(* Logix 5000 project; controller Hose_HP_Test_Rig_V1 vendor 1 type 14 code 149 rev 32.11; software revision 32.00 *)
// Hose HP Test Rig - 4 Station

TASK MainTask (continuous, watchdog 500 ms) : MainProgram

MODULES
   Local : vendor 1 type 14 code 149 (Compact 0, rev 32.11)
       : 1769-IQ32 (Compact 2, rev 3.1, Input RPI 20 ms)
      Discrete_IO : Embedded (Compact 1, rev 3.1, Output RPI 20 ms)
       : vendor 1 type 7 code 73 (Compact 3, rev 3.1, Output RPI 20 ms)
       : 1769-IF8 (Compact 5, rev 1.1, Output RPI 80 ms)
       : 1769-IF8 (Compact 4, rev 1.1, Output RPI 80 ms)
      VERIFYPLC : vendor 1 type 14 code 196 (Ethernet 192.168.4.180, rev 32.1, $d488c7ae$ RPI 20 ms, $26341d39$ RPI 20 ms, $f5226f78$ RPI 20 ms, $c4b3cc1b$ RPI 20 ms, $dea25812$ RPI 20 ms, $98b97a8d$ RPI 20 ms, $11873bfc$ RPI 20 ms, $408f890f$ RPI 20 ms, $f2f849b6$ RPI 20 ms, $8edf7c21$ RPI 20 ms, $0545c3c0$ RPI 20 ms, $be141c43$ RPI 20 ms, $2e1c7de5$ RPI 20 ms, $86533d27$ RPI 20 ms, $ac6396f9$ RPI 20 ms, $0a9383db$ RPI 20 ms)
      REM : vendor 1534 type 12 code 8 (Ethernet 192.168.4.224, rev 1.1, StandardDataDriven RPI 5 ms)
END_MODULES

ADD_ON_INSTRUCTION BOTTOM_DECLAMP   (* revision 1.0 *)
VAR_INPUT
   SET_SEQ_NO : DINT; {required}
END_VAR
VAR_IN_OUT
   CUR_SEQ_NO : DINT; {required}
END_VAR
VAR_OUTPUT
   BOTTOM_DECLAMP_AUTO : BOOL; {required}
END_VAR
VAR_INPUT
   BOTTOM_CLAMP_PS : BOOL; {required}
END_VAR
VAR_OUTPUT
   BOTTOM_DECLAMP_OK : BOOL; {required}
END_VAR
VAR_INPUT
   BOTTOM_NOT_DECLAMPED : BOOL; {required}
   FAULTED : BOOL; {required}
   RST_SEQ_ON : BOOL; {required}
   NEXT_SEQ_NO : DINT; {required}
END_VAR
VAR
   BOTTOM_DECLAMP_SEQ_AUTO : BOOL; {access None}
   ONS1 : BOOL; {access None}
   BOTTOM_DECLAMP_CHK_DEL : TIMER := (PRE := 500); {access None}
END_VAR

ROUTINE Logic   (* ladder *)
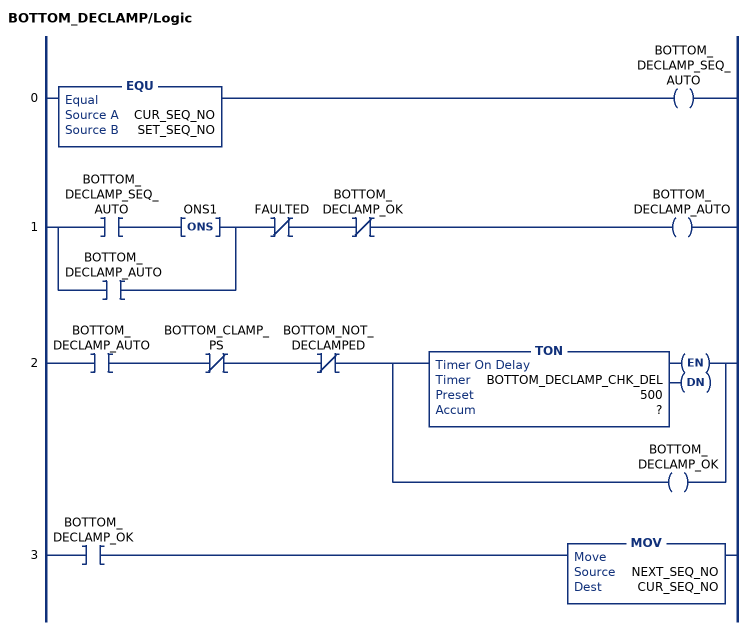
   0: EQU(CUR_SEQ_NO,SET_SEQ_NO)OTE(BOTTOM_DECLAMP_SEQ_AUTO);
   1: [XIC(BOTTOM_DECLAMP_SEQ_AUTO) ONS(ONS1) ,XIC(BOTTOM_DECLAMP_AUTO) ]XIO(FAULTED)XIO(BOTTOM_DECLAMP_OK)OTE(BOTTOM_DECLAMP_AUTO);
   2: XIC(BOTTOM_DECLAMP_AUTO)XIO(BOTTOM_CLAMP_PS)XIO(BOTTOM_NOT_DECLAMPED)[TON(BOTTOM_DECLAMP_CHK_DEL,?,?) ,OTE(BOTTOM_DECLAMP_OK) ];
   3: XIC(BOTTOM_DECLAMP_OK)MOV(NEXT_SEQ_NO,CUR_SEQ_NO);
END_ROUTINE
END_ADD_ON_INSTRUCTION

ADD_ON_INSTRUCTION CLAMP_FAULT   (* revision 1.0 *)
VAR_INPUT
   CLAMP_PR_SEL : BOOL; {required}
   CLAMP_PR_CHK : BOOL; {required}
   CLAMP_PR : DINT; {required}
   CLAMP_2BAR_LL : REAL; {required}
   CLAMP_2BAR_HL : REAL; {required}
   CLAMP_4BAR_LL : REAL; {required}
   CLAMP_4BAR_HL : REAL; {required}
   FLT_CLR_ONS : BOOL; {required}
END_VAR
VAR_OUTPUT
   CLAMP_2BPR_LOW : BOOL; {access Read Only, required}
   CLAMP_2BPR_HIGH : BOOL; {access Read Only, required}
   CLAMP_4BPR_LOW : BOOL; {access Read Only, required}
   CLAMP_4BPR_HIGH : BOOL; {access Read Only, required}
END_VAR
VAR_IN_OUT
   MSG : DINT; {required}
END_VAR

ROUTINE Logic   (* ladder *)
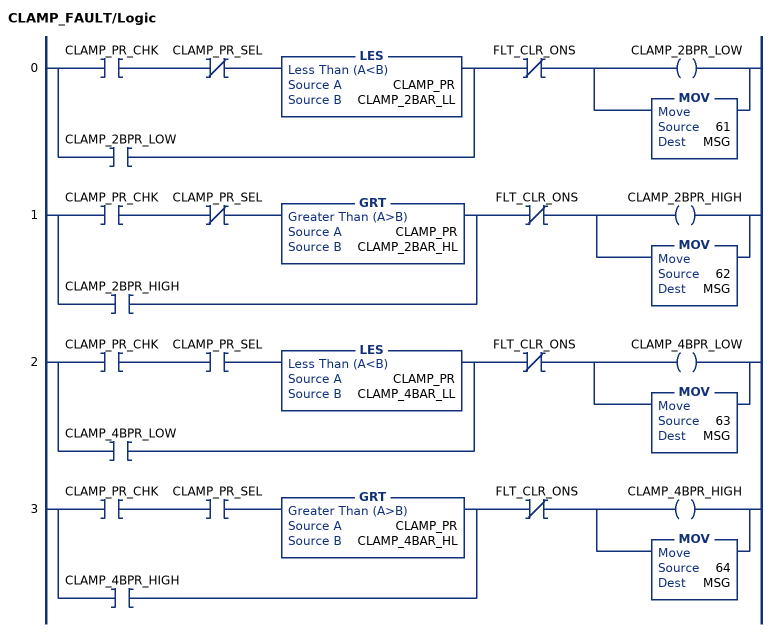
   0: [XIC(CLAMP_PR_CHK) XIO(CLAMP_PR_SEL) LES(CLAMP_PR,CLAMP_2BAR_LL) ,XIC(CLAMP_2BPR_LOW) ]XIO(FLT_CLR_ONS)[OTE(CLAMP_2BPR_LOW) ,MOV(61,MSG) ];
   1: [XIC(CLAMP_PR_CHK) XIO(CLAMP_PR_SEL) GRT(CLAMP_PR,CLAMP_2BAR_HL) ,XIC(CLAMP_2BPR_HIGH) ]XIO(FLT_CLR_ONS)[OTE(CLAMP_2BPR_HIGH) ,MOV(62,MSG) ];
   2: [XIC(CLAMP_PR_CHK) XIC(CLAMP_PR_SEL) LES(CLAMP_PR,CLAMP_4BAR_LL) ,XIC(CLAMP_4BPR_LOW) ]XIO(FLT_CLR_ONS)[OTE(CLAMP_4BPR_LOW) ,MOV(63,MSG) ];
   3: [XIC(CLAMP_PR_CHK) XIC(CLAMP_PR_SEL) GRT(CLAMP_PR,CLAMP_4BAR_HL) ,XIC(CLAMP_4BPR_HIGH) ]XIO(FLT_CLR_ONS)[OTE(CLAMP_4BPR_HIGH) ,MOV(64,MSG) ];
END_ROUTINE
END_ADD_ON_INSTRUCTION

ADD_ON_INSTRUCTION CONSTRICTION_FILL_OFF_SEQ   (* revision 1.0 *)
VAR_INPUT
   SET_SEQ_NO : DINT; {required}
END_VAR
VAR_IN_OUT
   CURR_SEQ_NO : DINT; {required}
END_VAR
VAR_INPUT
   TEST_ON : BOOL; {required}
END_VAR
VAR_OUTPUT
   CFILL_VAL_OFF : BOOL; {required}
   EXHS_VAL_OFF : BOOL; {required}
END_VAR
VAR_INPUT
   FAULTED : BOOL; {required}
   RST_SEQ_ON : BOOL; {required}
   NEXT_SEQ_NO : DINT; {required}
END_VAR
VAR
   SEQ_START : BOOL; {access None}
   ONS1 : BOOL; {access None}
   CFILL_VAL_OFF_DEL : TIMER := (PRE := 500); {access None}
   ONS2 : BOOL; {access None}
   ONS3 : BOOL; {access None}
END_VAR

ROUTINE Logic   (* ladder *)
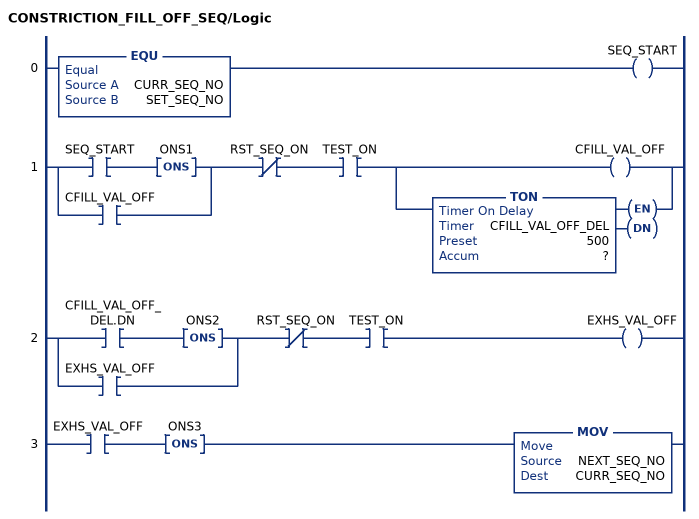
   0: EQU(CURR_SEQ_NO,SET_SEQ_NO)OTE(SEQ_START);
   1: [XIC(SEQ_START) ONS(ONS1) ,XIC(CFILL_VAL_OFF) ]XIO(RST_SEQ_ON)XIC(TEST_ON)[OTE(CFILL_VAL_OFF) ,TON(CFILL_VAL_OFF_DEL,?,?) ];
   2: [XIC(CFILL_VAL_OFF_DEL.DN) ONS(ONS2) ,XIC(EXHS_VAL_OFF) ]XIO(RST_SEQ_ON)XIC(TEST_ON)OTE(EXHS_VAL_OFF);
   3: XIC(EXHS_VAL_OFF)ONS(ONS3)MOV(NEXT_SEQ_NO,CURR_SEQ_NO);
END_ROUTINE
END_ADD_ON_INSTRUCTION

ADD_ON_INSTRUCTION CONSTRICTION_FILL_ON_SEQ   (* revision 1.0 *)
VAR_INPUT
   SET_SEQ_NO : DINT; {required}
END_VAR
VAR_IN_OUT
   CURR_SEQ_NO : DINT; {required}
END_VAR
VAR_INPUT
   TEST_STS : DINT; {required}
END_VAR
VAR_OUTPUT
   EXHS_VAL_ON : BOOL; {required}
   CFILL_VAL_ON : BOOL; {required}   // CONSTRICTION FILL VALVE ON
END_VAR
VAR_INPUT
   CFILL_VAL_OFF : BOOL; {required}
   RST_SEQ_ON : BOOL; {required}
   RST_EXHS_VAL_OFF : BOOL; {required}
   EXHS_VAL_OFF : BOOL; {required}
   FAULTED : BOOL; {required}
   NEXT_SEQ_NO : DINT; {required}
END_VAR
VAR
   SEQ_START : BOOL; {access None}
   ONS1 : BOOL; {access None}
   CFILL_VAL_ON_DEL : TIMER := (PRE := 500); {access None}
   ONS2 : BOOL; {access None}
   ONS3 : BOOL; {access None}
END_VAR

ROUTINE Logic   (* ladder *)
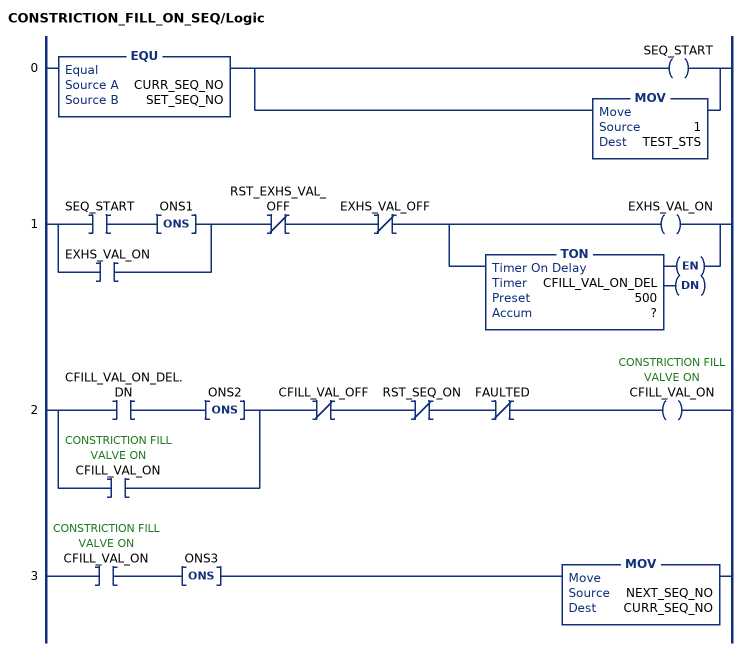
   0: EQU(CURR_SEQ_NO,SET_SEQ_NO)[OTE(SEQ_START) ,MOV(1,TEST_STS) ];
   1: [XIC(SEQ_START) ONS(ONS1) ,XIC(EXHS_VAL_ON) ]XIO(RST_EXHS_VAL_OFF)XIO(EXHS_VAL_OFF)[OTE(EXHS_VAL_ON) ,TON(CFILL_VAL_ON_DEL,?,?) ];
   2: [XIC(CFILL_VAL_ON_DEL.DN) ONS(ONS2) ,XIC(CFILL_VAL_ON) ]XIO(CFILL_VAL_OFF)XIO(RST_SEQ_ON)XIO(FAULTED)OTE(CFILL_VAL_ON);
   3: XIC(CFILL_VAL_ON)ONS(ONS3)MOV(NEXT_SEQ_NO,CURR_SEQ_NO);
END_ROUTINE
END_ADD_ON_INSTRUCTION

ADD_ON_INSTRUCTION DA_SOL_FWD_SEQ   (* revision 1.0 *)
VAR_IN_OUT
   DA_SOL_SEQ : DINT; {required}
END_VAR
VAR_OUTPUT
   DA_SOL_SOL : BOOL; {required}
END_VAR
VAR_INPUT
   DA_SOL_PS : BOOL; {required}
END_VAR
VAR_OUTPUT
   DA_PS_OK : BOOL; {required}
   DA_SOL_PS_FLT : BOOL; {required}
END_VAR
VAR_INPUT
   FAULT_CLEAR : BOOL; {required}
   RUN_CODE : DINT; {required}
END_VAR
VAR_IN_OUT
   MSG_CODE : DINT; {required}
END_VAR
VAR_INPUT
   FLT_CODE : DINT; {required}
END_VAR
VAR_IN_OUT
   ERROR_CODE : DINT; {required}
END_VAR
VAR_INPUT
   NEXT_SEQ_NO : DINT; {required}
END_VAR
VAR_IN_OUT
   ACT_SEQ_NO : DINT; {required}
END_VAR
VAR
   DA_SOL_PS_FAULT : TIMER := (PRE := 3000); {access None}
   DA_SOL_SEQ_ON : BOOL; {access Read Only}
   DA_SOL_PS_CHK : TIMER := (PRE := 500); {access None}
END_VAR

ROUTINE Logic   (* ladder *)
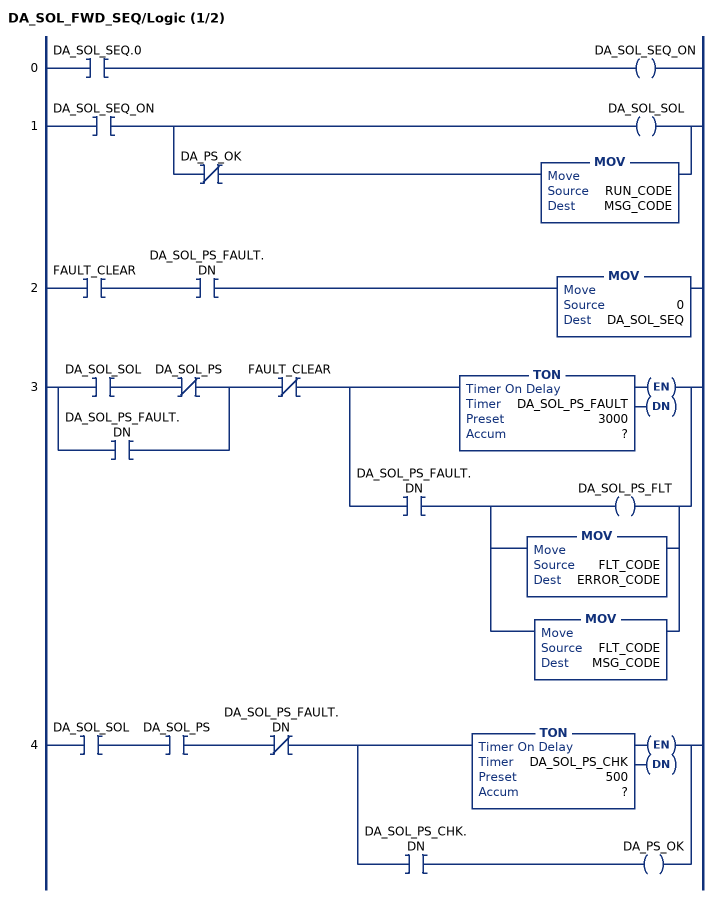
   0: XIC(DA_SOL_SEQ.0)OTE(DA_SOL_SEQ_ON);
   1: XIC(DA_SOL_SEQ_ON)[OTE(DA_SOL_SOL) ,XIO(DA_PS_OK) MOV(RUN_CODE,MSG_CODE) ];
   2: XIC(FAULT_CLEAR)XIC(DA_SOL_PS_FAULT.DN)MOV(0,DA_SOL_SEQ);
   3: [XIC(DA_SOL_SOL) XIO(DA_SOL_PS) ,XIC(DA_SOL_PS_FAULT.DN) ]XIO(FAULT_CLEAR)[TON(DA_SOL_PS_FAULT,?,?) ,XIC(DA_SOL_PS_FAULT.DN) [OTE(DA_SOL_PS_FLT) ,MOV(FLT_CODE,ERROR_CODE) ,MOV(FLT_CODE,MSG_CODE) ] ];
   4: XIC(DA_SOL_SOL)XIC(DA_SOL_PS)XIO(DA_SOL_PS_FAULT.DN)[TON(DA_SOL_PS_CHK,?,?) ,XIC(DA_SOL_PS_CHK.DN) OTE(DA_PS_OK) ];
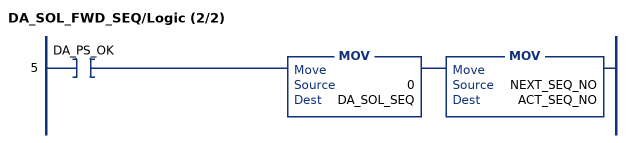
   5: XIC(DA_PS_OK)MOV(0,DA_SOL_SEQ)MOV(NEXT_SEQ_NO,ACT_SEQ_NO);
END_ROUTINE
END_ADD_ON_INSTRUCTION

ADD_ON_INSTRUCTION DA_SOL_RET_SEQ   (* revision 1.0 *)
VAR_IN_OUT
   DA_SOL_RET_SEQ : DINT; {required}
END_VAR
VAR_OUTPUT
   RET_SOL : BOOL; {required}
END_VAR
VAR_INPUT
   FWD_SOL_PS : BOOL; {required}
END_VAR
VAR_OUTPUT
   RET_SOL_PS_FLT : BOOL; {required}
END_VAR
VAR_INPUT
   FAULT_CLEAR : BOOL; {required}
   RUN_CODE : DINT; {required}
END_VAR
VAR_IN_OUT
   MSG_CODE : DINT; {required}
END_VAR
VAR_INPUT
   FLT_CODE : DINT; {required}
END_VAR
VAR_IN_OUT
   ERROR_CODE : DINT; {required}
END_VAR
VAR_INPUT
   SET_SEQ_NO : DINT; {required}
END_VAR
VAR_IN_OUT
   ACT_SEQ_NO : DINT; {required}
END_VAR
VAR
   DA_SOL_SEQ_ON : BOOL; {access None}
   DA_SOL_PS_FAULT : TIMER; {access None}
   RET_SOL_PS_FAULT : TIMER := (PRE := 3000); {access None}
   RET_SOL_PS_CHK : TIMER := (PRE := 500); {access None}
   RET_PS_OK : BOOL; {access None}
   ONS1 : BOOL; {access None}
END_VAR

ROUTINE Logic   (* ladder *)
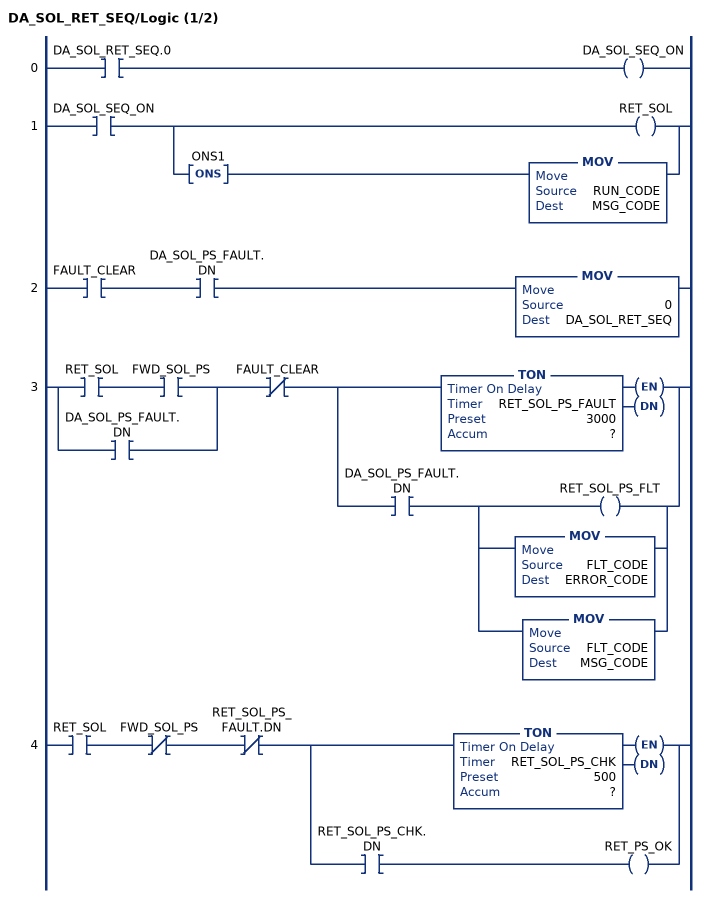
   0: XIC(DA_SOL_RET_SEQ.0)OTE(DA_SOL_SEQ_ON);
   1: XIC(DA_SOL_SEQ_ON)[OTE(RET_SOL) ,ONS(ONS1) MOV(RUN_CODE,MSG_CODE) ];
   2: XIC(FAULT_CLEAR)XIC(DA_SOL_PS_FAULT.DN)MOV(0,DA_SOL_RET_SEQ);
   3: [XIC(RET_SOL) XIC(FWD_SOL_PS) ,XIC(DA_SOL_PS_FAULT.DN) ]XIO(FAULT_CLEAR)[TON(RET_SOL_PS_FAULT,?,?) ,XIC(DA_SOL_PS_FAULT.DN) [OTE(RET_SOL_PS_FLT) ,MOV(FLT_CODE,ERROR_CODE) ,MOV(FLT_CODE,MSG_CODE) ] ];
   4: XIC(RET_SOL)XIO(FWD_SOL_PS)XIO(RET_SOL_PS_FAULT.DN)[TON(RET_SOL_PS_CHK,?,?) ,XIC(RET_SOL_PS_CHK.DN) OTE(RET_PS_OK) ];
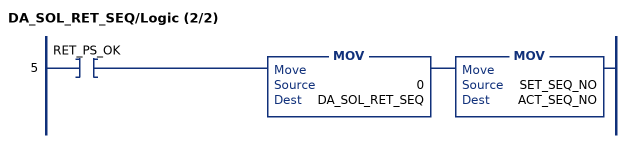
   5: XIC(RET_PS_OK)MOV(0,DA_SOL_RET_SEQ)MOV(SET_SEQ_NO,ACT_SEQ_NO);
END_ROUTINE
END_ADD_ON_INSTRUCTION

ADD_ON_INSTRUCTION DOOR_CLOSE   (* revision 1.0 *)
VAR_INPUT
   SET_SEQ_NO : DINT; {required}
END_VAR
VAR_IN_OUT
   CUR_SEQ_NO : DINT; {required}
END_VAR
VAR_INPUT
   LH_START_PB : BOOL; {required}
END_VAR
VAR_OUTPUT
   DOOR_CLOSE_OK_AUTO : BOOL; {required}
END_VAR
VAR_INPUT
   DOOR_NOT_CLOSED : BOOL; {required}
   DOOR_OPEN_RS : BOOL; {required}
END_VAR
VAR_OUTPUT
   DOOR_CLOSE_ABORT : BOOL; {required}
END_VAR
VAR_INPUT
   FAULTED : BOOL; {required}
   NEXT_SEQ_NO : DINT; {required}
END_VAR
VAR_IN_OUT
   DOOR_CLOSE_STS : DINT; {required}
END_VAR
VAR
   DOOR_CLOSE_SEQ_START : BOOL; {access None}
   ONS1 : BOOL; {access None}
   DUMMIT : BOOL; {access None}
END_VAR

ROUTINE Logic   (* ladder *)
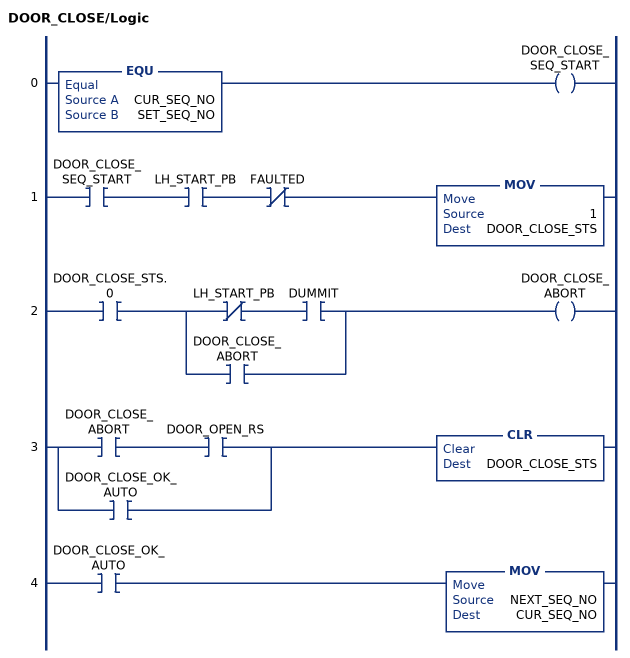
   0: EQU(CUR_SEQ_NO,SET_SEQ_NO)OTE(DOOR_CLOSE_SEQ_START);
   1: XIC(DOOR_CLOSE_SEQ_START)XIC(LH_START_PB)XIO(FAULTED)MOV(1,DOOR_CLOSE_STS);
   2: XIC(DOOR_CLOSE_STS.0)[XIO(LH_START_PB) XIC(DUMMIT) ,XIC(DOOR_CLOSE_ABORT) ]OTE(DOOR_CLOSE_ABORT);
   3: [XIC(DOOR_CLOSE_ABORT) XIC(DOOR_OPEN_RS) ,XIC(DOOR_CLOSE_OK_AUTO) ]CLR(DOOR_CLOSE_STS);
   4: XIC(DOOR_CLOSE_OK_AUTO)MOV(NEXT_SEQ_NO,CUR_SEQ_NO);
END_ROUTINE
END_ADD_ON_INSTRUCTION

ADD_ON_INSTRUCTION DROP_CHECK   (* revision 1.0 *)
VAR_INPUT
   SET_SEQ_NO : DINT; {required}
END_VAR
VAR_IN_OUT
   CURR_SEQ_NO : DINT; {required}
END_VAR
VAR_INPUT
   COMPARE_TIMER_SET_TIME : REAL; {required}
END_VAR
VAR_OUTPUT
   ACT_TIME : REAL; {required}
END_VAR
VAR_INPUT
   ACT_PR : REAL; {required}
   P1 : REAL; {required}
   PR_DIFF_LL : REAL; {required}
   PR_DIFF_HL : REAL; {required}
END_VAR
VAR_OUTPUT
   ACT_DROP : REAL; {required}
   DROP_OK : BOOL; {required}
   DROP_NOK : BOOL; {required}
END_VAR
VAR_INPUT
   CLR_FAIL_ONS : BOOL; {required}
   RUN_CODE : DINT; {visible}
   PASS_CODE : DINT; {required}
   FLT_CODE : DINT; {required}
END_VAR
VAR_IN_OUT
   ERR_CODE : DINT; {required}
   MSG_CODE : DINT; {required}
END_VAR
VAR_INPUT
   INITIALISE : BOOL; {required}
   ABORT : BOOL; {required}
   NEXT_SEQ_NO : DINT; {required}
END_VAR
VAR_OUTPUT
   P2 : REAL; {access None, required}
END_VAR
VAR
   COMPARE_TIMER : TIMER; {access None}
   DUMMIT : BOOL; {access None}
END_VAR

ROUTINE Logic   (* ladder *)
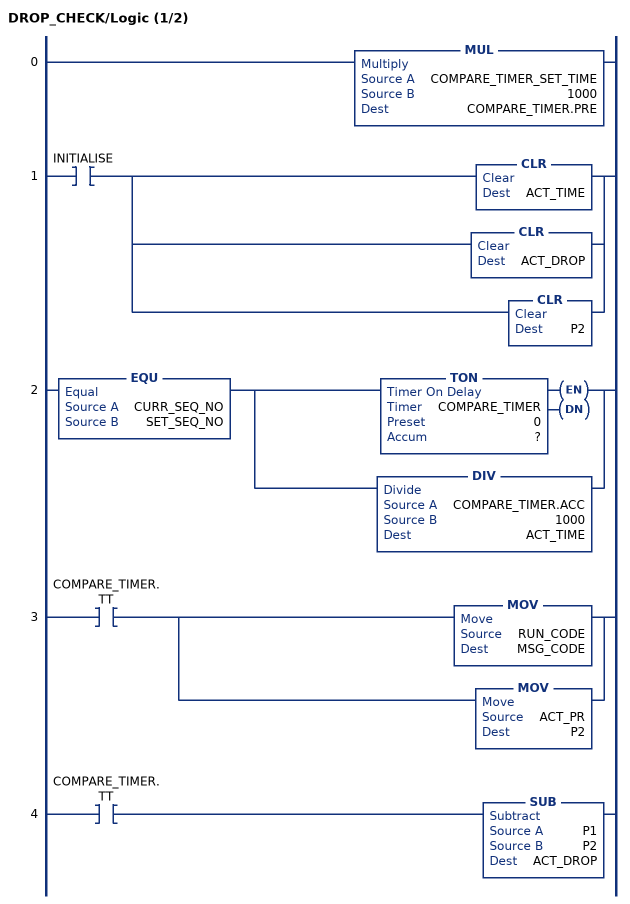
   0: MUL(COMPARE_TIMER_SET_TIME,1000,COMPARE_TIMER.PRE);
   1: XIC(INITIALISE)[CLR(ACT_TIME) ,CLR(ACT_DROP) ,CLR(P2) ];
   2: EQU(CURR_SEQ_NO,SET_SEQ_NO)[TON(COMPARE_TIMER,?,?) ,DIV(COMPARE_TIMER.ACC,1000,ACT_TIME) ];
   3: XIC(COMPARE_TIMER.TT)[MOV(RUN_CODE,MSG_CODE) ,MOV(ACT_PR,P2) ];
   4: XIC(COMPARE_TIMER.TT)SUB(P1,P2,ACT_DROP);
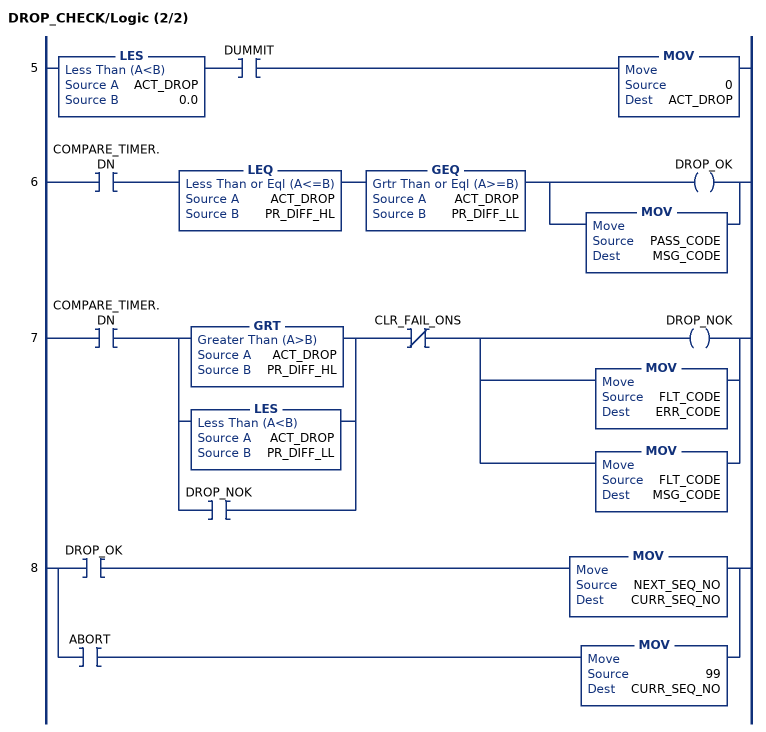
   5: LES(ACT_DROP,0.0)XIC(DUMMIT)MOV(0,ACT_DROP);
   6: XIC(COMPARE_TIMER.DN)LEQ(ACT_DROP,PR_DIFF_HL)GEQ(ACT_DROP,PR_DIFF_LL)[OTE(DROP_OK) ,MOV(PASS_CODE,MSG_CODE) ];
   7: XIC(COMPARE_TIMER.DN)[[GRT(ACT_DROP,PR_DIFF_HL) ,LES(ACT_DROP,PR_DIFF_LL) ] ,XIC(DROP_NOK) ]XIO(CLR_FAIL_ONS)[OTE(DROP_NOK) ,MOV(FLT_CODE,ERR_CODE) ,MOV(FLT_CODE,MSG_CODE) ];
   8: [XIC(DROP_OK) MOV(NEXT_SEQ_NO,CURR_SEQ_NO) ,XIC(ABORT) MOV(99,CURR_SEQ_NO) ];
END_ROUTINE
END_ADD_ON_INSTRUCTION

ADD_ON_INSTRUCTION Fill_Stab_Flt_Msg   (* revision 1.0 *)
VAR_INPUT
   LOW_STN : BOOL; {required}
   HIGH_STN : BOOL; {required}
   LOW_FLT_FAIL_CODE : DINT; {required}
   HIGH_FLT_FAIL_CODE : DINT; {required}
END_VAR
VAR_IN_OUT
   MSG_STN : DINT; {required}
END_VAR

ROUTINE Logic   (* ladder *)
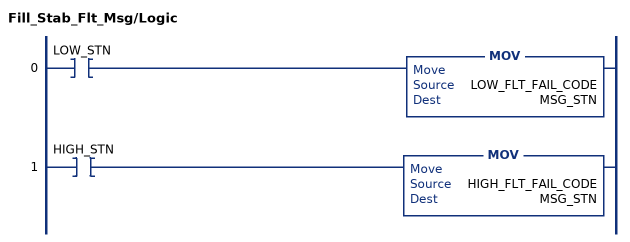
   0: XIC(LOW_STN)MOV(LOW_FLT_FAIL_CODE,MSG_STN);
   1: XIC(HIGH_STN)MOV(HIGH_FLT_FAIL_CODE,MSG_STN);
END_ROUTINE
END_ADD_ON_INSTRUCTION

ADD_ON_INSTRUCTION FILL_VAL_OFF   (* revision 1.0 *)
VAR_INPUT
   SET_SEQ_NO : DINT; {required}
END_VAR
VAR_IN_OUT
   ACT_SEQ_NO : DINT; {required}
END_VAR
VAR_OUTPUT
   TEST_VAL_OFF : BOOL; {required}
END_VAR
VAR_INPUT
   FAULTED : BOOL; {required}
   NEXT_SEQ_NO : DINT; {required}
END_VAR
VAR
   NEXT_SEQ_DEL : TIMER := (PRE := 500); {access None}
END_VAR

ROUTINE Logic   (* ladder *)
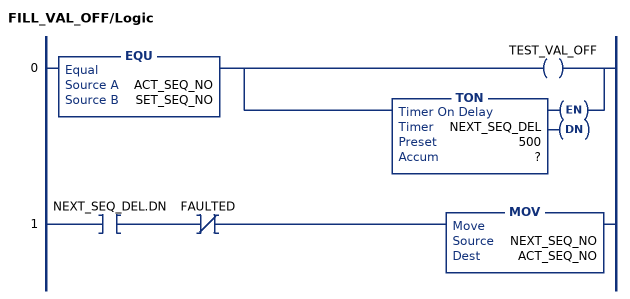
   0: EQU(ACT_SEQ_NO,SET_SEQ_NO)[OTE(TEST_VAL_OFF) ,TON(NEXT_SEQ_DEL,?,?) ];
   1: XIC(NEXT_SEQ_DEL.DN)XIO(FAULTED)MOV(NEXT_SEQ_NO,ACT_SEQ_NO);
END_ROUTINE
END_ADD_ON_INSTRUCTION

ADD_ON_INSTRUCTION INIT_CYCLE   (* revision 1.0 *)

ROUTINE Logic   (* ladder *)
END_ROUTINE
END_ADD_ON_INSTRUCTION

ADD_ON_INSTRUCTION PR_CHECK   (* revision 1.0 *)
// Revision note:
// PR FILL TIME->CHECK LIM->NEXT
VAR_INPUT
   SET_SEQ : DINT; {required}
END_VAR
VAR_IN_OUT
   CURR_SEQ : DINT; {required}
END_VAR
VAR_INPUT
   ACT_PR : REAL; {required}
   PR_LL : REAL; {required}
   PR_HL : REAL; {required}
   SET_TIME : REAL; {required}
END_VAR
VAR_OUTPUT
   ACT_TIME : REAL; {required}
   LIMIT_LOW : BOOL; {access None, required}
   LIMIT_HIGH : BOOL; {required}
   PR_AT_END : REAL; {required}
END_VAR
VAR_INPUT
   CLEAR_ACTUALS : BOOL; {required}
   CLEAR_ERROR : BOOL; {required}
   ABORT : BOOL; {required}
   SEQ_STS_CODE : DINT; {required}
END_VAR
VAR_IN_OUT
   TEST_STS : DINT; {required}
END_VAR
VAR_INPUT
   RUN_CODE : DINT; {required}
END_VAR
VAR_IN_OUT
   MSG_CODE : DINT; {required}
END_VAR
VAR_INPUT
   LIM_LOW_CODE : DINT; {required}
   LIM_HIGH_CODE : DINT; {required}
END_VAR
VAR_IN_OUT
   ERR_CODE : DINT; {required}
END_VAR
VAR_INPUT
   NEXT_SEQ_NO : DINT; {required}
END_VAR
VAR
   COMPARE_TIMER : TIMER; {access None}
   LIMIT_OK : BOOL; {access None}
   ONS1 : BOOL; {access None}
END_VAR

ROUTINE Logic   (* ladder *)
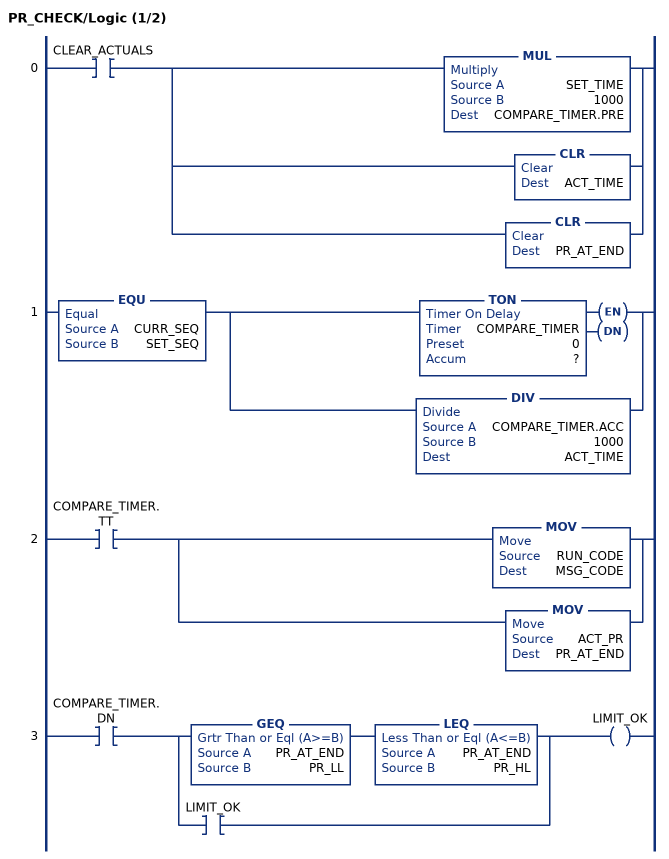
   0: XIC(CLEAR_ACTUALS)[MUL(SET_TIME,1000,COMPARE_TIMER.PRE) ,CLR(ACT_TIME) ,CLR(PR_AT_END) ];
   1: EQU(CURR_SEQ,SET_SEQ)[TON(COMPARE_TIMER,?,?) ,DIV(COMPARE_TIMER.ACC,1000,ACT_TIME) ];
   2: XIC(COMPARE_TIMER.TT)[MOV(RUN_CODE,MSG_CODE) ,MOV(ACT_PR,PR_AT_END) ];
   3: XIC(COMPARE_TIMER.DN)[GEQ(PR_AT_END,PR_LL) LEQ(PR_AT_END,PR_HL) ,XIC(LIMIT_OK) ]OTE(LIMIT_OK);
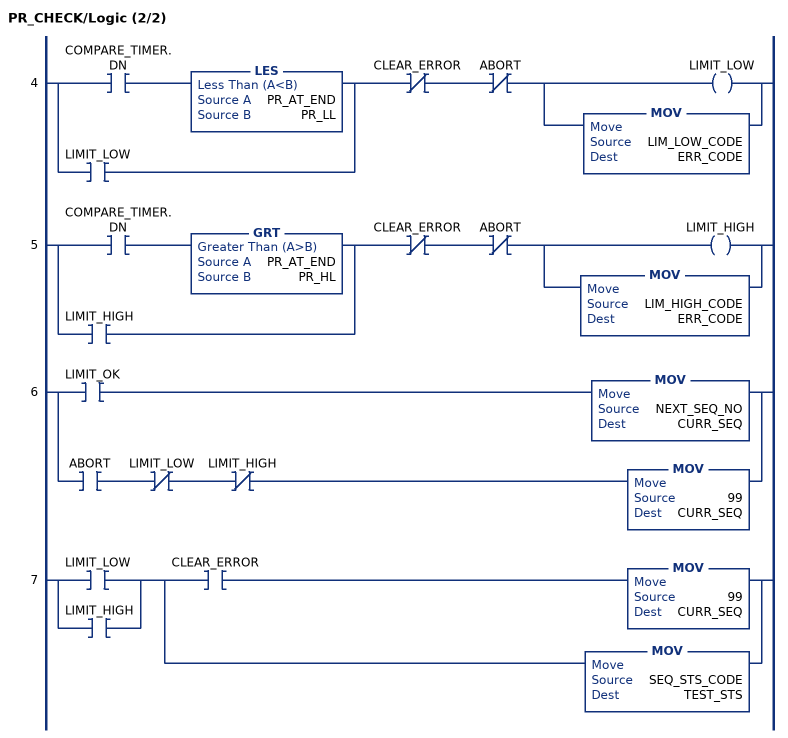
   4: [XIC(COMPARE_TIMER.DN) LES(PR_AT_END,PR_LL) ,XIC(LIMIT_LOW) ]XIO(CLEAR_ERROR)XIO(ABORT)[OTE(LIMIT_LOW) ,MOV(LIM_LOW_CODE,ERR_CODE) ];
   5: [XIC(COMPARE_TIMER.DN) GRT(PR_AT_END,PR_HL) ,XIC(LIMIT_HIGH) ]XIO(CLEAR_ERROR)XIO(ABORT)[OTE(LIMIT_HIGH) ,MOV(LIM_HIGH_CODE,ERR_CODE) ];
   6: [XIC(LIMIT_OK) MOV(NEXT_SEQ_NO,CURR_SEQ) ,XIC(ABORT) XIO(LIMIT_LOW) XIO(LIMIT_HIGH) MOV(99,CURR_SEQ) ];
   7: [XIC(LIMIT_LOW) ,XIC(LIMIT_HIGH) ][XIC(CLEAR_ERROR) MOV(99,CURR_SEQ) ,MOV(SEQ_STS_CODE,TEST_STS) ];
END_ROUTINE
END_ADD_ON_INSTRUCTION

ADD_ON_INSTRUCTION Rst_Seq_On   (* revision 1.0 *)
VAR_INPUT
   FAULTED : BOOL; {required}
   FAILED : BOOL; {required}
   INPUT_1_16 : DINT; {required}
        .10   // DOOR OPEN RS
        .11   // FAIL RST KS
        .12   // TOP CLAMP PS
        .13   // BOTTOM CLAMP PS
        .6   // EMG STOP PB
        .7   // FAULT RESET PB
END_VAR
VAR_OUTPUT
   FLT_CLR_ONS : BOOL; {required}
END_VAR
VAR_INPUT
   SET_MODE_SEL : BOOL; {required}
   FAIL_LAMP : BOOL; {required}
   FAIL_RST_ONS : BOOL; {required}
   INDV_OFF : BOOL; {required}
   EMG_FAULT : BOOL; {required}
END_VAR
VAR_OUTPUT
   RST_SEQ_ON : BOOL; {required}
   RST_TEST_VAL_OFF : BOOL; {required}
   PR_EXHS_OK : BOOL; {required}
   RST_SEQ_OVER : BOOL; {required}
END_VAR
VAR_INPUT
   FAIL_BIN_FULL : BOOL; {required}
   TOP_CLAMP_PT_FAULT : BOOL; {required}
   BOTTOM_CLAMP_PT_FAULT : BOOL; {required}
END_VAR
VAR_IN_OUT
   ACT_PR : REAL; {required}
END_VAR
VAR_INPUT
   PR_EXHS_LIMIT : REAL; {required}
   FAIL_BIN_SEQ : INT; {required}
END_VAR
VAR_IN_OUT
   MSG : DINT; {required}
   CURR_SEQ_NO : DINT; {required}
END_VAR
VAR
   ONS1 : BOOL; {access None}
   ONS2 : BOOL; {access None}
   ONS74 : BOOL; {access None}
   RST_SEQ_OVER_DEL : TIMER := (PRE := 500); {access None}
   FLT_RST_ONS : BOOL;
   SEQ_NO_SET : DINT;
   ONS3 : BOOL; {access None}
   ONS4 : BOOL; {access None}
   RST_EXHS_OFF_DEL : TIMER := (PRE := 500); {access None}
   ONS5 : BOOL; {access None}
END_VAR

ROUTINE Logic   (* ladder *)
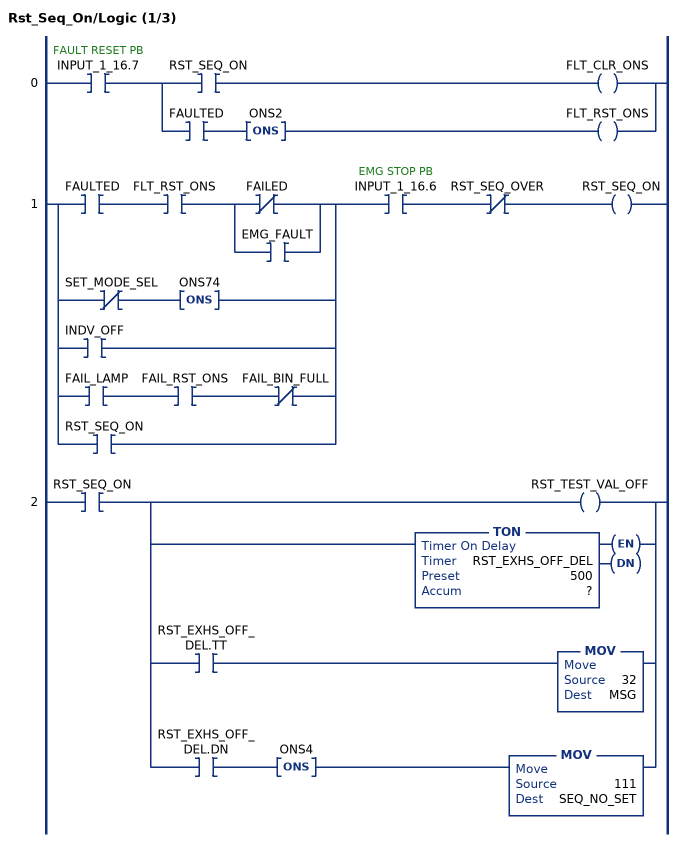
   0: XIC(INPUT_1_16.7)[XIC(RST_SEQ_ON) OTE(FLT_CLR_ONS) ,XIC(FAULTED) ONS(ONS2) OTE(FLT_RST_ONS) ];
   1: [XIC(FAULTED) XIC(FLT_RST_ONS) [XIO(FAILED) ,XIC(EMG_FAULT) ] ,XIO(SET_MODE_SEL) ONS(ONS74) ,XIC(INDV_OFF) ,XIC(FAIL_LAMP) XIC(FAIL_RST_ONS) XIO(FAIL_BIN_FULL) ,XIC(RST_SEQ_ON) ]XIC(INPUT_1_16.6)XIO(RST_SEQ_OVER)OTE(RST_SEQ_ON);
   2: XIC(RST_SEQ_ON)[OTE(RST_TEST_VAL_OFF) ,TON(RST_EXHS_OFF_DEL,?,?) ,XIC(RST_EXHS_OFF_DEL.TT) MOV(32,MSG) ,XIC(RST_EXHS_OFF_DEL.DN) ONS(ONS4) MOV(111,SEQ_NO_SET) ];
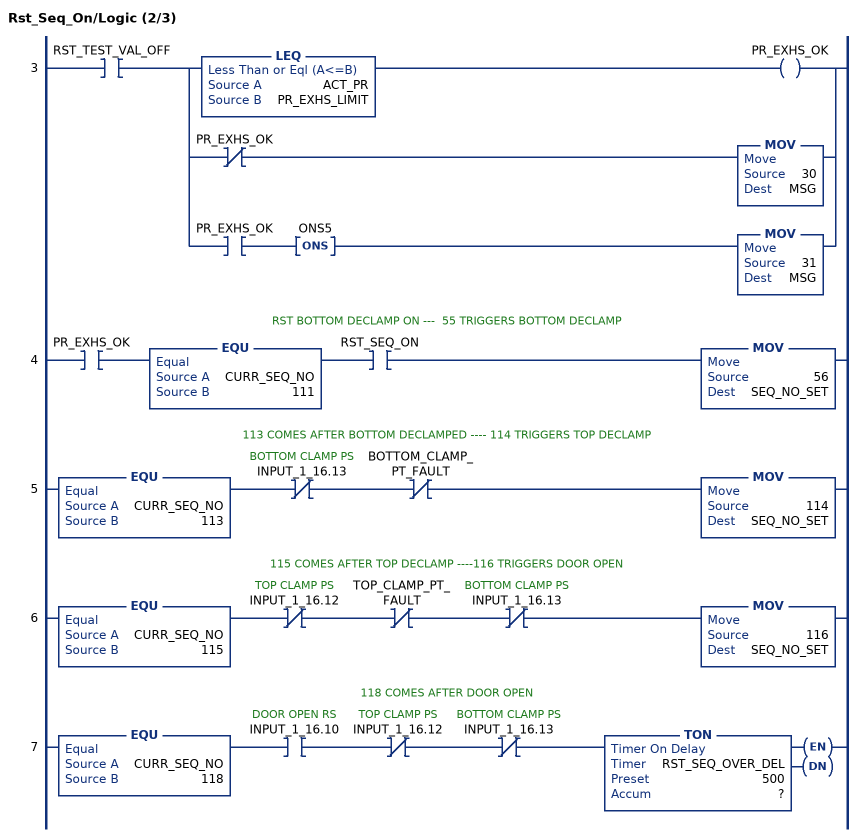
   3: XIC(RST_TEST_VAL_OFF)[LEQ(ACT_PR,PR_EXHS_LIMIT) OTE(PR_EXHS_OK) ,XIO(PR_EXHS_OK) MOV(30,MSG) ,XIC(PR_EXHS_OK) ONS(ONS5) MOV(31,MSG) ];
   // RST BOTTOM DECLAMP ON ---  55 TRIGGERS BOTTOM DECLAMP
   4: XIC(PR_EXHS_OK)EQU(CURR_SEQ_NO,111)XIC(RST_SEQ_ON)MOV(56,SEQ_NO_SET);
   // 113 COMES AFTER BOTTOM DECLAMPED ---- 114 TRIGGERS TOP DECLAMP
   5: EQU(CURR_SEQ_NO,113)XIO(INPUT_1_16.13)XIO(BOTTOM_CLAMP_PT_FAULT)MOV(114,SEQ_NO_SET);
   // 115 COMES AFTER TOP DECLAMP ----116 TRIGGERS DOOR OPEN
   6: EQU(CURR_SEQ_NO,115)XIO(INPUT_1_16.12)XIO(TOP_CLAMP_PT_FAULT)XIO(INPUT_1_16.13)MOV(116,SEQ_NO_SET);
   // 118 COMES AFTER DOOR OPEN
   7: EQU(CURR_SEQ_NO,118)XIC(INPUT_1_16.10)XIO(INPUT_1_16.12)XIO(INPUT_1_16.13)TON(RST_SEQ_OVER_DEL,?,?);
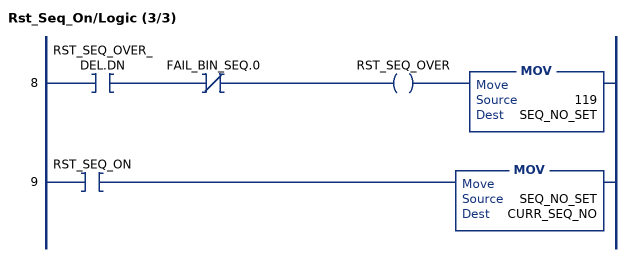
   8: XIC(RST_SEQ_OVER_DEL.DN)XIO(FAIL_BIN_SEQ.0)OTE(RST_SEQ_OVER)MOV(119,SEQ_NO_SET);
   9: XIC(RST_SEQ_ON)MOV(SEQ_NO_SET,CURR_SEQ_NO);
END_ROUTINE
END_ADD_ON_INSTRUCTION
